// TIA Portal V20 export
TYPE "typeCmControlNodeSoftCam"
// stored: Namespace Unit1.Em5
   STRUCT
      transferPnPLeftAxisX : "Unit1.Em5.typeCmControlNodeSoftCamtransferPnPLeftAxisX";
      transferPnPLeftAxisY : "Unit1.Em5.typeCmControlNodeSoftCamtransferPnPLeftAxisY";
      transferPnPLeftAxisZ : "Unit1.Em5.typeCmControlNodeSoftCamtransferPnPLeftAxisZ";
      transferPnPRightAxisX : "Unit1.Em5.typeCmControlNodeSoftCamtransferPnPRightAxisX";
      transferPnPRightAxisY : "Unit1.Em5.typeCmControlNodeSoftCamtransferPnPRightAxisY";
      transferPnPRightAxisZ : "Unit1.Em5.typeCmControlNodeSoftCamtransferPnPRightAxisZ";
   END_STRUCT;
END_TYPE
